// TIA Portal project "ACTEA_Ex6" (V15.1)

(* hardware
DEVICE "S7-1200 station_2"  S7-1200 Station
   slot 0: "Rack_0"  S7-1200 Rack  Rack  V1.0
   slot 1: "PLC_1"  CPU 1214C DC/DC/DC  6ES7 214-1AG31-0XB0  V3.0
   slot 3: "AQ 1x12BIT_1"  AQ1 signal board  6ES7 232-4HA30-0XB0  V1.0
*)

// ===== PLC "PLC_1"  CPU 1214C DC/DC/DC =====

VAR_GLOBAL   // PLC tag table "Tag-Table"
   "System_Byte" AT %MB254 : Byte;
   "FirstScan" AT %M254.0 : Bool;
   "DiagStatusUpdate" AT %M254.1 : Bool;
   "AlwaysTRUE" AT %M254.2 : Bool;
   "AlwaysFALSE" AT %M254.3 : Bool;
   "Clock_Byte" AT %MB255 : Byte;
   "Clock_10Hz" AT %M255.0 : Bool;
   "Clock_5Hz" AT %M255.1 : Bool;
   "Clock_2.5Hz" AT %M255.2 : Bool;
   "Clock_2Hz" AT %M255.3 : Bool;
   "Clock_1.25Hz" AT %M255.4 : Bool;
   "Clock_1Hz" AT %M255.5 : Bool;
   "Clock_0.625Hz" AT %M255.6 : Bool;
   "Clock_0.5Hz" AT %M255.7 : Bool;
   "iCC_BtnStop_S1" AT %I0.0 : Bool;   // Stop button
   "iCC_BtnStart_S2" AT %I0.2 : Bool;   // Start button
   "iCC_RlyEms_KES" AT %I1.0 : Bool;   // Safety relay OK
   "iCC_McbMot_QM1" AT %I1.1 : Bool;   // Motor circuit breaker
   "iCC_ConMot_KM1" AT %I1.2 : Bool;   // Feedback signal contactor
   "oCC_LmpStart_H1" AT %Q0.0 : Bool;   // Lamp start
   "oCC_LmpStop_H3" AT %Q0.2 : Bool;   // Lamp stop
   "oCC_ConMot_KM1" AT %Q0.6 : Bool;   // Contactor motor
   "mMotStarted" AT %M0.0 : Bool;   // Motor started
END_VAR

VAR_GLOBAL CONSTANT   // PLC tag table "Tag-Table"
   "None" : Pip := 65535;
   "Automatic update" : Pip := 0;
   "PIP 1" : Pip := 1;
   "PIP 2" : Pip := 2;
   "PIP 3" : Pip := 3;
   "PIP 4" : Pip := 4;
   "PIP OB Servo" : Pip := 32768;
   "Local~MC" : Hw_SubModule := 51;
   "Local~Common" : Hw_SubModule := 50;
   "Local~Device" : Hw_Device := 32;
   "Local~Configuration" : Hw_SubModule := 33;
   "Local~Exec" : Hw_SubModule := 52;
   "Local(1)" : Hw_SubModule := 49;
   "Local~PROFINET_interface_1(1)" : Hw_Interface := 64;
   "Local~PROFINET_interface_1~Port_1(1)" : Hw_Interface := 65;
   "Local~HSC_1(1)" : Hw_Hsc := 257;
   "Local~HSC_2(1)" : Hw_Hsc := 258;
   "Local~HSC_3(1)" : Hw_Hsc := 259;
   "Local~HSC_4(1)" : Hw_Hsc := 260;
   "Local~HSC_5(1)" : Hw_Hsc := 261;
   "Local~HSC_6(1)" : Hw_Hsc := 262;
   "Local~AI_2_1(1)" : Hw_SubModule := 263;
   "Local~DI_14_DQ_10_1(1)" : Hw_SubModule := 264;
   "Local~Pulse_1(1)" : Hw_Pwm := 265;
   "Local~Pulse_2(1)" : Hw_Pwm := 266;
   "Local~Pulse_3(1)" : Hw_Pwm := 267;
   "Local~Pulse_4(1)" : Hw_Pwm := 268;
   "OB_Main(1)" : OB_PCYCLE := 1;
END_VAR

FUNCTION "FC_DOL_EMS" : Void   // FC1, FBD
{ S7_Optimized_Access := 'TRUE' }
VERSION : 0.1
BEGIN

REGION Network 1: Start-stop circuit "mMotStarted"
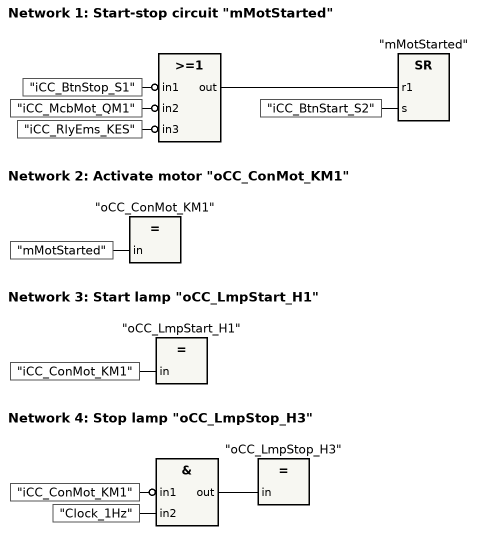
   IF "iCC_BtnStart_S2" THEN
       "mMotStarted" := TRUE;   // SR flip-flop
   END_IF;
   IF NOT "iCC_BtnStop_S1" OR NOT "iCC_McbMot_QM1" OR NOT "iCC_RlyEms_KES" THEN
       "mMotStarted" := FALSE;
   END_IF;
END_REGION

REGION Network 2: Activate motor "oCC_ConMot_KM1"
   "oCC_ConMot_KM1" := "mMotStarted";
END_REGION

REGION Network 3: Start lamp "oCC_LmpStart_H1"
   "oCC_LmpStart_H1" := "iCC_ConMot_KM1";
END_REGION

REGION Network 4: Stop lamp "oCC_LmpStop_H3"
   "oCC_LmpStop_H3" := NOT "iCC_ConMot_KM1" AND "Clock_1Hz";
END_REGION
END_FUNCTION

ORGANIZATION_BLOCK "Main"   // OB1, LAD, ProgramCycle
TITLE = "Main Program Sweep (Cycle)"
{ S7_Optimized_Access := 'TRUE' }
VERSION : 0.1
   VAR_INPUT
      Initial_Call : Bool;   // Initial call of this OB
      Remanence : Bool;   // =True, if remanent data are available
   END_VAR
BEGIN

REGION Network 1
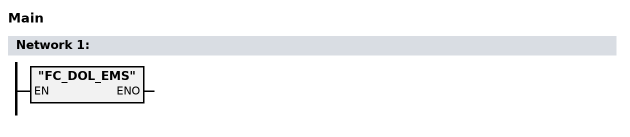
   RUNG wire#powerrail
      "FC_DOL_EMS"()
   END_RUNG
   // the same network as SCL:
   "FC_DOL_EMS"();
END_REGION
END_ORGANIZATION_BLOCK